// TIA Portal project "激光打标_V15.1" (V15.1)

(* hardware
DEVICE "S7-1200 station_1"  S7-1200 Station
   slot 0: "Rack_0"  S7-1200 Rack  Rack  V1.0
   slot 1: "A170648_14 CPU  1214C"  CPU 1214C DC/DC/DC  6ES7 214-1AG40-0XB0  V4.2
   slot 2: "DI 16x24VDC/DQ 16xRelay_1"  SM 1223 DI16/DQ16 x relay  6ES7 223-1PL32-0XB0  V2.0
   slot 3: "DI 16x24VDC/DQ 16xRelay_2"  SM 1223 DI16/DQ16 x relay  6ES7 223-1PL32-0XB0  V2.0
*)

// ===== PLC "A170648_14 CPU  1214C"  CPU 1214C DC/DC/DC =====

VAR_GLOBAL   // PLC tag table "默认变量表"
   "启动" AT %I0.0 : Bool;
   "复位" AT %I0.1 : Bool;
   "安全门" AT %I0.2 : Bool;
   "急停" AT %I0.3 : Bool;
   "气源检测" AT %I0.4 : Bool;
   "手自动" AT %I0.5 : Bool;
   "激光打码完成" AT %I0.6 : Bool;
   "激光打码报警" AT %I0.7 : Bool;
   "1#升降按钮" AT %I1.0 : Bool;
   "1#气爪松紧按钮" AT %I1.1 : Bool;
   "1#固定按钮" AT %I1.2 : Bool;
   "2#升降按钮" AT %I1.3 : Bool;
   "2#气爪松紧按钮" AT %I1.4 : Bool;
   "2#固定按钮" AT %I1.5 : Bool;
   "工件在位" AT %I2.0 : Bool;
   "防护门上限位" AT %I2.1 : Bool;
   "防护门下限位" AT %I2.2 : Bool;
   "工装移栽进到位" AT %I2.3 : Bool;
   "工装移栽退到位" AT %I2.4 : Bool;
   "备用(2)" AT %I2.5 : Bool;
   "备用(4)" AT %I2.6 : Bool;
   "备用(3)" AT %I2.7 : Bool;
   "1#固定进到位" AT %I3.0 : Bool;
   "1#固定退到位" AT %I3.1 : Bool;
   "备用" AT %I3.2 : Bool;
   "1#左气爪松开到位" AT %I3.3 : Bool;
   "备用(1)" AT %I3.4 : Bool;
   "1#右气爪松开到位" AT %I3.5 : Bool;
   "1#机械手升到位" AT %I3.6 : Bool;
   "1#机械手降到位" AT %I3.7 : Bool;
   "2#机械手升到位" AT %I4.0 : Bool;
   "2#机械手降到位" AT %I4.1 : Bool;
   "备用(31)" AT %I4.2 : Bool;
   "2#左气爪松开到位" AT %I4.3 : Bool;
   "备用(32)" AT %I4.4 : Bool;
   "2#右气爪松开到位" AT %I4.5 : Bool;
   "2#固定进到位" AT %I4.6 : Bool;
   "2#固定退到位" AT %I4.7 : Bool;
   "备用(5)" AT %I5.0 : Bool;
   "备用(6)" AT %I5.1 : Bool;
   "备用(7)" AT %I5.2 : Bool;
   "备用(8)" AT %I5.3 : Bool;
   "备用(9)" AT %I5.4 : Bool;
   "备用(10)" AT %I5.5 : Bool;
   "备用(11)" AT %I5.6 : Bool;
   "备用(12)" AT %I5.7 : Bool;
   "启动打标" AT %Q0.0 : Bool;
   "备用(13)" AT %Q0.1 : Bool;
   "三色灯——红" AT %Q0.2 : Bool;
   "三色灯——黄" AT %Q0.3 : Bool;
   "三色灯——绿" AT %Q0.4 : Bool;
   "三色灯——蜂鸣器" AT %Q0.5 : Bool;
   "气源开关" AT %Q0.6 : Bool;
   "备用(14)" AT %Q0.7 : Bool;
   "合格指示灯" AT %Q1.0 : Bool;
   "不合格指示灯" AT %Q1.1 : Bool;
   "防护门上升" AT %Q2.0 : Bool;
   "防护门下降" AT %Q2.1 : Bool;
   "工装移载前进" AT %Q2.2 : Bool;
   "工装移载后退" AT %Q2.3 : Bool;
   "备用(15)" AT %Q2.4 : Bool;
   "备用(16)" AT %Q2.5 : Bool;
   "备用(17)" AT %Q2.6 : Bool;
   "备用(18)" AT %Q2.7 : Bool;
   "1#机械手上升" AT %Q3.0 : Bool;
   "1#机械手下降" AT %Q3.1 : Bool;
   "1#机械手气爪夹紧" AT %Q3.2 : Bool;
   "1#机械手气爪松开" AT %Q3.3 : Bool;
   "备用(19)" AT %Q3.4 : Bool;
   "备用(20)" AT %Q3.5 : Bool;
   "1#固定气缸进" AT %Q3.6 : Bool;
   "1#固定气缸退" AT %Q3.7 : Bool;
   "2#机械手上升" AT %Q4.0 : Bool;
   "2#机械手下降" AT %Q4.1 : Bool;
   "2#机械手气爪夹紧" AT %Q4.2 : Bool;
   "2#机械手气爪松开" AT %Q4.3 : Bool;
   "备用(21)" AT %Q4.4 : Bool;
   "备用(22)" AT %Q4.5 : Bool;
   "2#固定气缸进" AT %Q4.6 : Bool;
   "2#固定气缸退" AT %Q4.7 : Bool;
   "备用(23)" AT %Q5.0 : Bool;
   "备用(24)" AT %Q5.1 : Bool;
   "备用(25)" AT %Q5.2 : Bool;
   "备用(26)" AT %Q5.3 : Bool;
   "备用(27)" AT %Q5.4 : Bool;
   "备用(28)" AT %Q5.5 : Bool;
   "备用(29)" AT %Q5.6 : Bool;
   "备用(30)" AT %Q5.7 : Bool;
   "程序停止" AT %M100.0 : Bool;
   "复位完成" AT %M100.1 : Bool;
   "Clock_1Hz" AT %M0.5 : Bool;
   "Tag_1" AT %M100.3 : Bool;
   "AlwaysFALSE" AT %M1.3 : Bool;
   "Tag_2" AT %M30.0 : Bool;
   "Clock_Byte" AT %MB0 : Byte;
   "Clock_10Hz" AT %M0.0 : Bool;
   "Clock_5Hz" AT %M0.1 : Bool;
   "Clock_2.5Hz" AT %M0.2 : Bool;
   "Clock_2Hz" AT %M0.3 : Bool;
   "Clock_1.25Hz" AT %M0.4 : Bool;
   "Clock_0.625Hz" AT %M0.6 : Bool;
   "Clock_0.5Hz" AT %M0.7 : Bool;
   "System_Byte" AT %MB1 : Byte;
   "FirstScan" AT %M1.0 : Bool;
   "DiagStatusUpdate" AT %M1.1 : Bool;
   "AlwaysTRUE" AT %M1.2 : Bool;
   "Tag_3" AT %M300.0 : Bool;
   "Tag_4" AT %M300.4 : Bool;
   "Tag_5" AT %M300.1 : Bool;
   "Tag_6" AT %M300.5 : Bool;
   "Tag_7" AT %M300.3 : Bool;
   "Tag_8" AT %M300.7 : Bool;
   "Tag_9" AT %M312.0 : Bool;
   "Tag_10" AT %M3000.0 : Bool;
   "Tag_11" AT %M3000.1 : Bool;
   "Tag_12" AT %MD3004 : DWord;
   "Tag_13" AT %M3000.2 : Bool;
   "Tag_14" AT %M3000.3 : Bool;
   "Tag_15" AT %MW3004 : Word;
   "Tag_16" AT %M312.1 : Bool;
   "Tag_17" AT %M200.0 : Bool;
   "Tag_18" AT %M200.6 : Bool;
   "Tag_19" AT %M200.7 : Bool;
   "吸尘器" AT %MB10 : SInt;
END_VAR

DATA_BLOCK "SERVER"   // DB1
{ S7_Optimized_Access := 'FALSE' }
VERSION : 0.1
   VAR
      设备状态 : Int := 0;
      产品型号 : Int := 0;
      错误代码 : Int := 0;
      生产结果 : Int := 0;
      设备编号 : Int := 0;
      吸尘器 : Int;
   END_VAR
BEGIN
END_DATA_BLOCK

DATA_BLOCK "MB_TCON"   // DB2
{ S7_Optimized_Access := 'FALSE' }
VERSION : 0.1
   VAR
      MB_TCON : TCON_IP_v4;
   END_VAR
BEGIN
   MB_TCON.InterfaceId := 64;
   MB_TCON.ID := 1;
   MB_TCON.LocalPort := 502;
   MB_TCON.RemoteAddress.ADDR[1] := 0;
   MB_TCON.RemoteAddress.ADDR[2] := 0;
   MB_TCON.RemoteAddress.ADDR[3] := 0;
   MB_TCON.RemoteAddress.ADDR[4] := 0;
END_DATA_BLOCK

DATA_BLOCK "RESET_DB"   // DB3
{ S7_Optimized_Access := 'TRUE' }
VERSION : 0.1
// stored: InstanceOfName RESET
"RESET"
BEGIN
END_DATA_BLOCK

DATA_BLOCK "ALARM_DB"   // DB4
{ S7_Optimized_Access := 'TRUE' }
VERSION : 0.1
// stored: InstanceOfName ALARM
"ALARM"
BEGIN
END_DATA_BLOCK

DATA_BLOCK "1# jixieshou_DB"   // DB8
{ S7_Optimized_Access := 'TRUE' }
VERSION : 0.1
// stored: InstanceOfName 1# jixieshou
"1# jixieshou"
BEGIN
END_DATA_BLOCK

DATA_BLOCK "2#jixieshou_DB"   // DB9
{ S7_Optimized_Access := 'TRUE' }
VERSION : 0.1
// stored: InstanceOfName 2#jixieshou
"2#jixieshou"
BEGIN
END_DATA_BLOCK

DATA_BLOCK "AUTO_DB"   // DB10
{ S7_Optimized_Access := 'TRUE' }
VERSION : 0.1
// stored: InstanceOfName AUTO
"AUTO"
BEGIN
END_DATA_BLOCK

// folder: System blocks/Program resources

DATA_BLOCK "IEC_Timer_0_DB"   // DB5
{ S7_Optimized_Access := 'TRUE' }
AUTHOR : Simatic
FAMILY : IEC
NAME : IEC_TMR
VERSION : 1.0
// stored: InstanceOfName IEC_TIMER
"IEC_TIMER"
BEGIN
END_DATA_BLOCK

DATA_BLOCK "IEC_Timer_0_DB_1"   // DB6
{ S7_Optimized_Access := 'TRUE' }
AUTHOR : Simatic
FAMILY : IEC
NAME : IEC_TMR
VERSION : 1.0
// stored: InstanceOfName IEC_TIMER
"IEC_TIMER"
BEGIN
END_DATA_BLOCK

DATA_BLOCK "IEC_Timer_0_DB_3"   // DB12
{ S7_Optimized_Access := 'TRUE' }
AUTHOR : Simatic
FAMILY : IEC
NAME : IEC_TMR
VERSION : 1.0
// stored: InstanceOfName IEC_TIMER
"IEC_TIMER"
BEGIN
END_DATA_BLOCK

// folder: (top level)

FUNCTION_BLOCK "ALARM"   // FB1, LAD
{ S7_Optimized_Access := 'TRUE' }
VERSION : 0.1
   VAR
      "Error-ID" : Word;
      TEmp : Array[0..3] of Bool;
      IEC_Timer_0_Instance : TON_TIME;
      IEC_Timer_0_Instance_1 : TON_TIME;
      IEC_Timer_0_Instance_2 : TON_TIME;
      IEC_Timer_0_Instance_3 : TON_TIME;
      IEC_Timer_0_Instance_4 : TON_TIME;
      IEC_Timer_0_Instance_5 : TON_TIME;
      IEC_Timer_0_Instance_6 : TON_TIME;
      IEC_Timer_0_Instance_7 : TON_TIME;
      IEC_Timer_0_Instance_8 : TON_TIME;
      IEC_Timer_0_Instance_9 : TON_TIME;
      IEC_Timer_0_Instance_10 : TON_TIME;
      IEC_Timer_0_Instance_11 : TON_TIME;
      IEC_Timer_0_Instance_12 : TON_TIME;
      IEC_Timer_0_Instance_13 : TON_TIME;
      IEC_Timer_0_Instance_14 : TON_TIME;
      "STEP" : Int;
      IEC_Timer_0_Instance_15 : TON_TIME;
      IEC_Timer_0_Instance_16 : TON_TIME;
   END_VAR
   VAR_TEMP   // added for the SCL form of the ladder/FBD networks
      _w1 : Bool;
   END_VAR
BEGIN

REGION Network 1
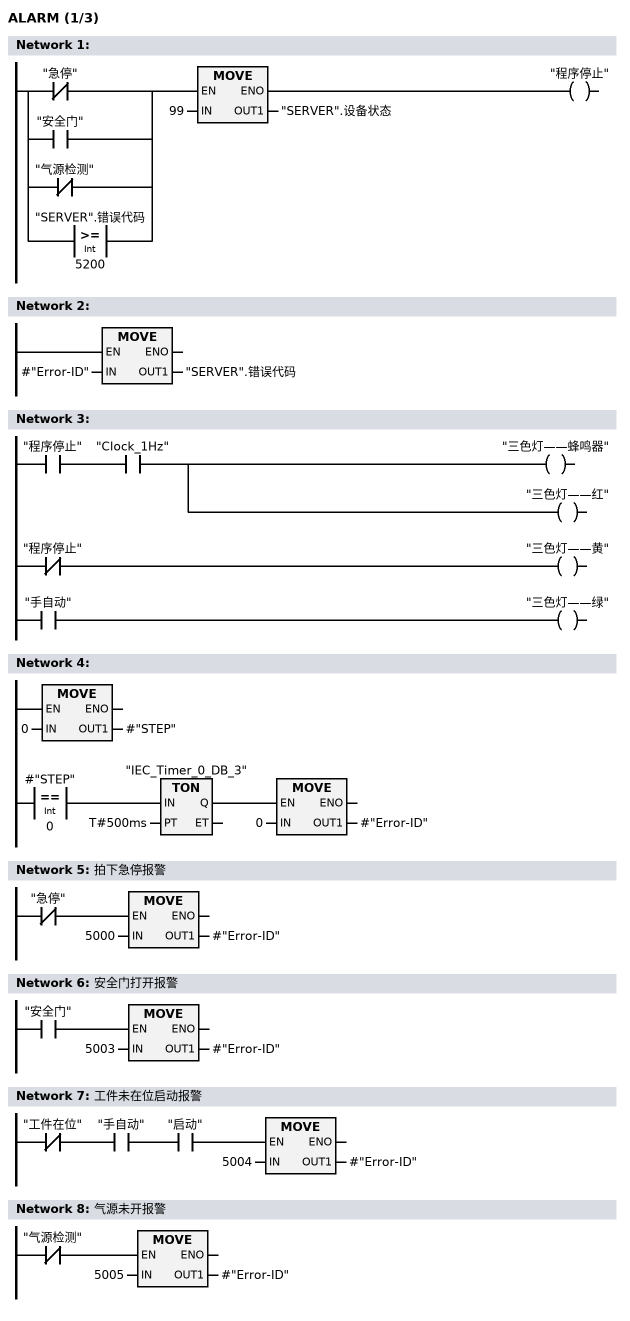
   RUNG wire#powerrail
      I_Contact( "急停" )
      wire#w1
      Move(in := 99, out1 => "SERVER".设备状态)
      Coil( "程序停止" )
   END_RUNG
   RUNG wire#powerrail
      Contact( "安全门" )
   END_RUNG wire#w1
   RUNG wire#powerrail
      I_Contact( "气源检测" )
   END_RUNG wire#w1
   RUNG wire#powerrail
      { S7_Templates := "SrcType := Int" } GE_Contact(in1 := "SERVER".错误代码, in2 := 5200)
   END_RUNG wire#w1
   // the same network as SCL:
   #_w1 := NOT "急停" OR "安全门" OR NOT "气源检测" OR ("SERVER".错误代码 >= 5200);
   IF #_w1 THEN "SERVER".设备状态 := 99; END_IF;
   "程序停止" := #_w1;
END_REGION

REGION Network 2
   RUNG wire#powerrail
      Move(in := #"Error-ID", out1 => "SERVER".错误代码)
   END_RUNG
   // the same network as SCL:
   "SERVER".错误代码 := #"Error-ID";
END_REGION

REGION Network 3
   RUNG wire#powerrail
      Contact( "程序停止" )
      Contact( "Clock_1Hz" )
      wire#w1
      Coil( "三色灯——蜂鸣器" )
   END_RUNG
   RUNG wire#w1
      Coil( "三色灯——红" )
   END_RUNG
   RUNG wire#powerrail
      I_Contact( "程序停止" )
      Coil( "三色灯——黄" )
   END_RUNG
   RUNG wire#powerrail
      Contact( "手自动" )
      Coil( "三色灯——绿" )
   END_RUNG
   // the same network as SCL:
   "三色灯——蜂鸣器" := "程序停止" AND "Clock_1Hz";
   "三色灯——红" := "三色灯——蜂鸣器";
   "三色灯——黄" := NOT "程序停止";
   "三色灯——绿" := "手自动";
END_REGION

REGION Network 4
   #"STEP" := 0;
   "IEC_Timer_0_DB_3".TON(IN := #"STEP" = 0, PT := T#500ms);
   IF "IEC_Timer_0_DB_3".Q THEN #"Error-ID" := 0; END_IF;
END_REGION

REGION Network 5: 拍下急停报警
   RUNG wire#powerrail
      I_Contact( "急停" )
      Move(in := 5000, out1 => #"Error-ID")
   END_RUNG
   // the same network as SCL:
   IF NOT "急停" THEN #"Error-ID" := 5000; END_IF;
END_REGION

REGION Network 6: 安全门打开报警
   RUNG wire#powerrail
      Contact( "安全门" )
      Move(in := 5003, out1 => #"Error-ID")
   END_RUNG
   // the same network as SCL:
   IF "安全门" THEN #"Error-ID" := 5003; END_IF;
END_REGION

REGION Network 7: 工件未在位启动报警
   RUNG wire#powerrail
      I_Contact( "工件在位" )
      Contact( "手自动" )
      Contact( "启动" )
      Move(in := 5004, out1 => #"Error-ID")
   END_RUNG
   // the same network as SCL:
   IF NOT "工件在位" AND "手自动" AND "启动" THEN #"Error-ID" := 5004; END_IF;
END_REGION

REGION Network 8: 气源未开报警
   RUNG wire#powerrail
      I_Contact( "气源检测" )
      Move(in := 5005, out1 => #"Error-ID")
   END_RUNG
   // the same network as SCL:
   IF NOT "气源检测" THEN #"Error-ID" := 5005; END_IF;
END_REGION

REGION Network 9: 工装移栽前进未到位报警
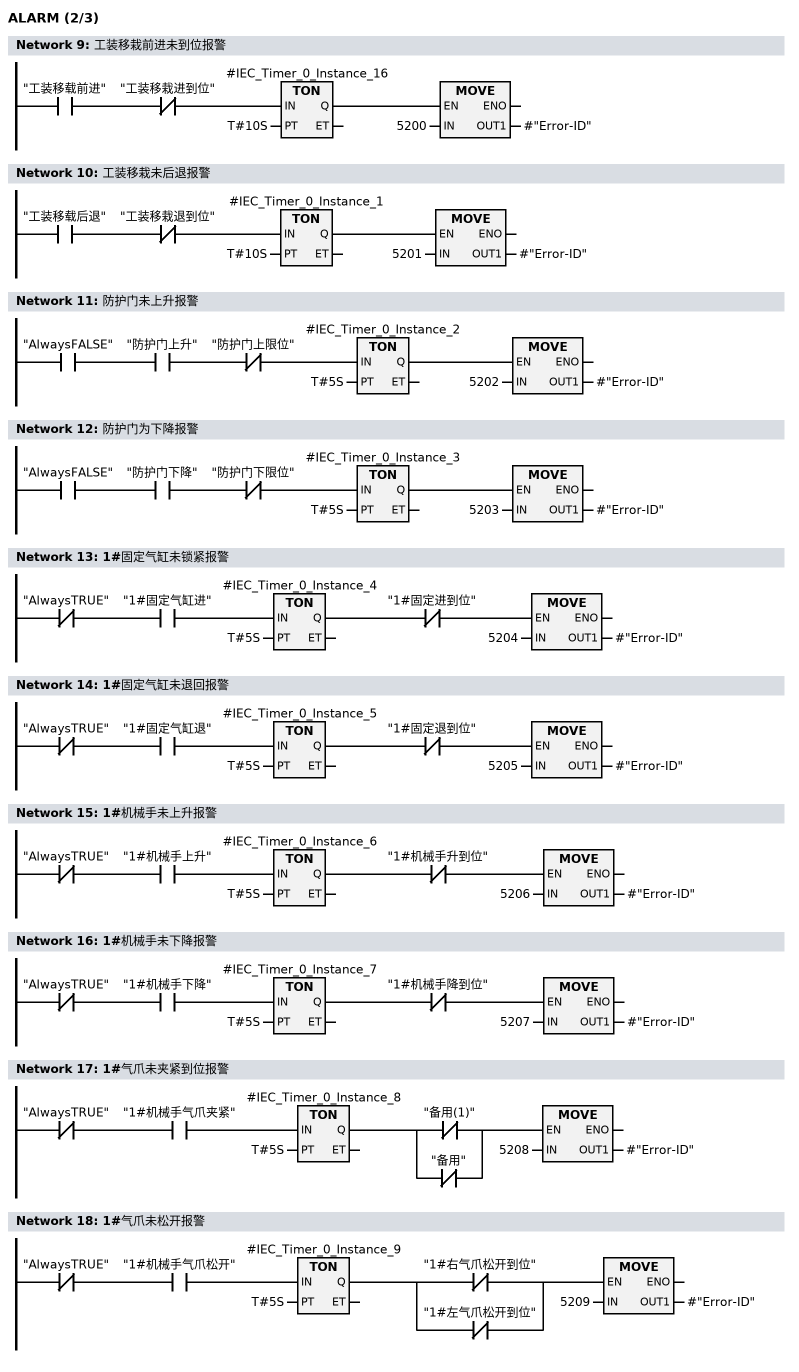
   #IEC_Timer_0_Instance_16(IN := "工装移载前进" AND NOT "工装移栽进到位", PT := T#10S);   // TON
   IF #IEC_Timer_0_Instance_16.Q THEN #"Error-ID" := 5200; END_IF;
END_REGION

REGION Network 10: 工装移栽未后退报警
   #IEC_Timer_0_Instance_1(IN := "工装移载后退" AND NOT "工装移栽退到位", PT := T#10S);   // TON
   IF #IEC_Timer_0_Instance_1.Q THEN #"Error-ID" := 5201; END_IF;
END_REGION

REGION Network 11: 防护门未上升报警
   #IEC_Timer_0_Instance_2(IN := "AlwaysFALSE" AND "防护门上升" AND NOT "防护门上限位", PT := T#5S);   // TON
   IF #IEC_Timer_0_Instance_2.Q THEN #"Error-ID" := 5202; END_IF;
END_REGION

REGION Network 12: 防护门为下降报警
   #IEC_Timer_0_Instance_3(IN := "AlwaysFALSE" AND "防护门下降" AND NOT "防护门下限位", PT := T#5S);   // TON
   IF #IEC_Timer_0_Instance_3.Q THEN #"Error-ID" := 5203; END_IF;
END_REGION

REGION Network 13: 1#固定气缸未锁紧报警
   #IEC_Timer_0_Instance_4(IN := NOT "AlwaysTRUE" AND "1#固定气缸进", PT := T#5S);   // TON
   IF #IEC_Timer_0_Instance_4.Q AND NOT "1#固定进到位" THEN #"Error-ID" := 5204; END_IF;
END_REGION

REGION Network 14: 1#固定气缸未退回报警
   #IEC_Timer_0_Instance_5(IN := NOT "AlwaysTRUE" AND "1#固定气缸退", PT := T#5S);   // TON
   IF #IEC_Timer_0_Instance_5.Q AND NOT "1#固定退到位" THEN #"Error-ID" := 5205; END_IF;
END_REGION

REGION Network 15: 1#机械手未上升报警
   #IEC_Timer_0_Instance_6(IN := NOT "AlwaysTRUE" AND "1#机械手上升", PT := T#5S);   // TON
   IF #IEC_Timer_0_Instance_6.Q AND NOT "1#机械手升到位" THEN #"Error-ID" := 5206; END_IF;
END_REGION

REGION Network 16: 1#机械手未下降报警
   #IEC_Timer_0_Instance_7(IN := NOT "AlwaysTRUE" AND "1#机械手下降", PT := T#5S);   // TON
   IF #IEC_Timer_0_Instance_7.Q AND NOT "1#机械手降到位" THEN #"Error-ID" := 5207; END_IF;
END_REGION

REGION Network 17: 1#气爪未夹紧到位报警
   #IEC_Timer_0_Instance_8(IN := NOT "AlwaysTRUE" AND "1#机械手气爪夹紧", PT := T#5S);   // TON
   IF #IEC_Timer_0_Instance_8.Q AND (NOT "备用(1)" OR NOT "备用") THEN #"Error-ID" := 5208; END_IF;
END_REGION

REGION Network 18: 1#气爪未松开报警
   #IEC_Timer_0_Instance_9(IN := NOT "AlwaysTRUE" AND "1#机械手气爪松开", PT := T#5S);   // TON
   IF #IEC_Timer_0_Instance_9.Q AND (NOT "1#右气爪松开到位" OR NOT "1#左气爪松开到位") THEN #"Error-ID" := 5209; END_IF;
END_REGION

REGION Network 19: 2#机械手未固定锁紧报警
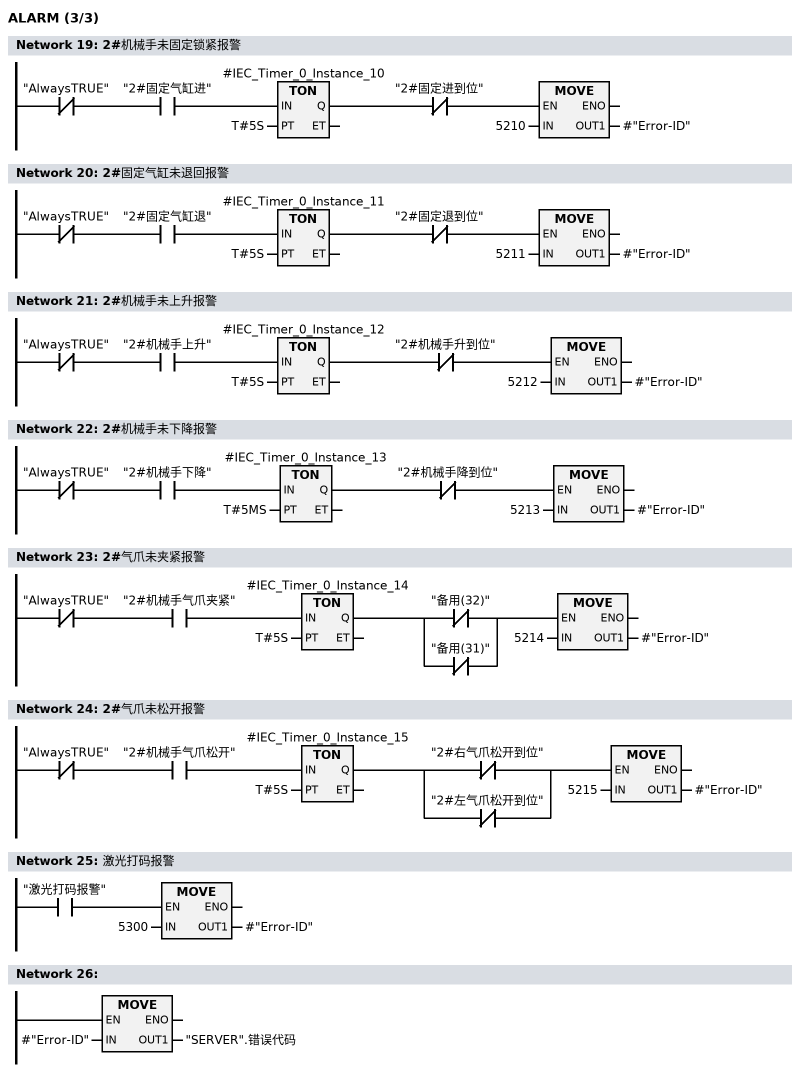
   #IEC_Timer_0_Instance_10(IN := NOT "AlwaysTRUE" AND "2#固定气缸进", PT := T#5S);   // TON
   IF #IEC_Timer_0_Instance_10.Q AND NOT "2#固定进到位" THEN #"Error-ID" := 5210; END_IF;
END_REGION

REGION Network 20: 2#固定气缸未退回报警
   #IEC_Timer_0_Instance_11(IN := NOT "AlwaysTRUE" AND "2#固定气缸退", PT := T#5S);   // TON
   IF #IEC_Timer_0_Instance_11.Q AND NOT "2#固定退到位" THEN #"Error-ID" := 5211; END_IF;
END_REGION

REGION Network 21: 2#机械手未上升报警
   #IEC_Timer_0_Instance_12(IN := NOT "AlwaysTRUE" AND "2#机械手上升", PT := T#5S);   // TON
   IF #IEC_Timer_0_Instance_12.Q AND NOT "2#机械手升到位" THEN #"Error-ID" := 5212; END_IF;
END_REGION

REGION Network 22: 2#机械手未下降报警
   #IEC_Timer_0_Instance_13(IN := NOT "AlwaysTRUE" AND "2#机械手下降", PT := T#5MS);   // TON
   IF #IEC_Timer_0_Instance_13.Q AND NOT "2#机械手降到位" THEN #"Error-ID" := 5213; END_IF;
END_REGION

REGION Network 23: 2#气爪未夹紧报警
   #IEC_Timer_0_Instance_14(IN := NOT "AlwaysTRUE" AND "2#机械手气爪夹紧", PT := T#5S);   // TON
   IF #IEC_Timer_0_Instance_14.Q AND (NOT "备用(32)" OR NOT "备用(31)") THEN #"Error-ID" := 5214; END_IF;
END_REGION

REGION Network 24: 2#气爪未松开报警
   #IEC_Timer_0_Instance_15(IN := NOT "AlwaysTRUE" AND "2#机械手气爪松开", PT := T#5S);   // TON
   IF #IEC_Timer_0_Instance_15.Q AND (NOT "2#右气爪松开到位" OR NOT "2#左气爪松开到位") THEN #"Error-ID" := 5215; END_IF;
END_REGION

REGION Network 25: 激光打码报警
   RUNG wire#powerrail
      Contact( "激光打码报警" )
      Move(in := 5300, out1 => #"Error-ID")
   END_RUNG
   // the same network as SCL:
   IF "激光打码报警" THEN #"Error-ID" := 5300; END_IF;
END_REGION

REGION Network 26
   RUNG wire#powerrail
      Move(in := #"Error-ID", out1 => "SERVER".错误代码)
   END_RUNG
   // the same network as SCL:
   "SERVER".错误代码 := #"Error-ID";
END_REGION
END_FUNCTION_BLOCK

FUNCTION_BLOCK "RESET"   // FB2, LAD
{ S7_Optimized_Access := 'TRUE' }
VERSION : 0.1
   VAR_INPUT
      Stop : Bool;
      Start : Bool;
   END_VAR
   VAR_OUTPUT
      Down : Bool;
   END_VAR
   VAR
      "Step" : Int;
   END_VAR
   VAR_TEMP   // added for the SCL form of the ladder/FBD networks
      _w1 : Bool;
   END_VAR
BEGIN

REGION Network 1
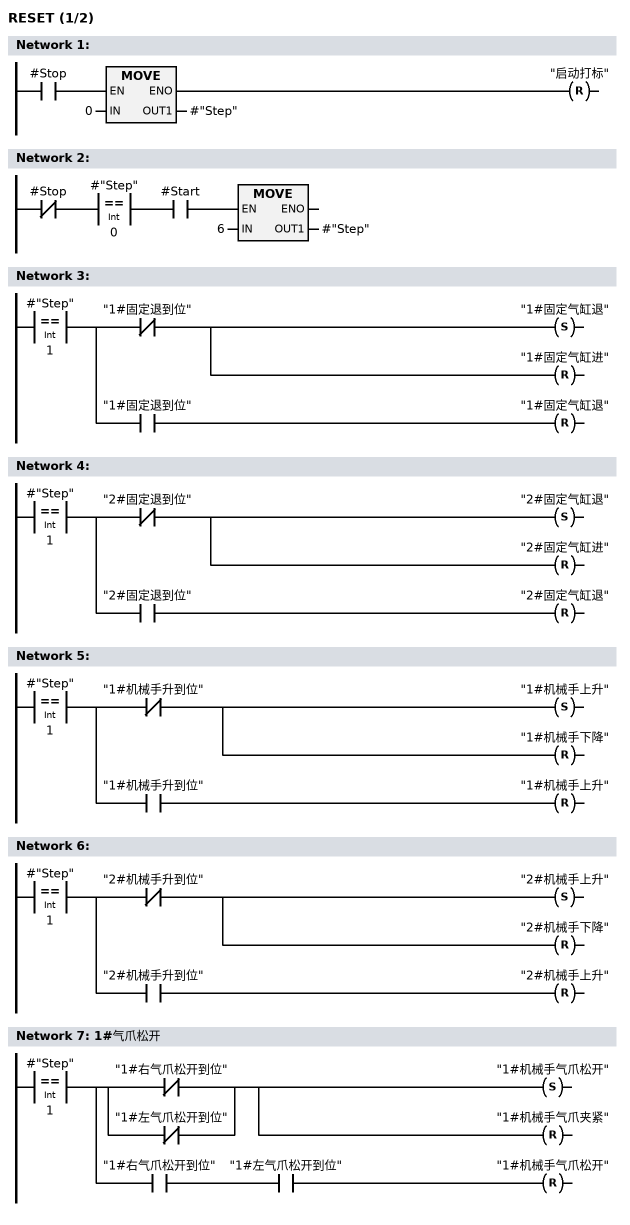
   RUNG wire#powerrail
      Contact( #Stop )
      Move(in := 0, out1 => #"Step")
      R_Coil( "启动打标" )
   END_RUNG
   // the same network as SCL:
   IF #Stop THEN
       #"Step" := 0;
       "启动打标" := FALSE;
   END_IF;
END_REGION

REGION Network 2
   RUNG wire#powerrail
      I_Contact( #Stop )
      { S7_Templates := "SrcType := Int" } EQ_Contact(in1 := #"Step", in2 := 0)
      Contact( #Start )
      Move(in := 6, out1 => #"Step")
   END_RUNG
   // the same network as SCL:
   IF NOT #Stop AND (#"Step" = 0) AND #Start THEN #"Step" := 6; END_IF;
END_REGION

REGION Network 3
   RUNG wire#powerrail
      { S7_Templates := "SrcType := Int" } EQ_Contact(in1 := #"Step", in2 := 1)
      wire#w1
      I_Contact( "1#固定退到位" )
      wire#w2
      S_Coil( "1#固定气缸退" )
   END_RUNG
   RUNG wire#w2
      R_Coil( "1#固定气缸进" )
   END_RUNG
   RUNG wire#w1
      Contact( "1#固定退到位" )
      R_Coil( "1#固定气缸退" )
   END_RUNG
   // the same network as SCL:
   #_w1 := #"Step" = 1;
   IF #_w1 AND NOT "1#固定退到位" THEN
       "1#固定气缸退" := TRUE;
       "1#固定气缸进" := FALSE;
   END_IF;
   IF #_w1 AND "1#固定退到位" THEN "1#固定气缸退" := FALSE; END_IF;
END_REGION

REGION Network 4
   RUNG wire#powerrail
      { S7_Templates := "SrcType := Int" } EQ_Contact(in1 := #"Step", in2 := 1)
      wire#w1
      I_Contact( "2#固定退到位" )
      wire#w2
      S_Coil( "2#固定气缸退" )
   END_RUNG
   RUNG wire#w2
      R_Coil( "2#固定气缸进" )
   END_RUNG
   RUNG wire#w1
      Contact( "2#固定退到位" )
      R_Coil( "2#固定气缸退" )
   END_RUNG
   // the same network as SCL:
   #_w1 := #"Step" = 1;
   IF #_w1 AND NOT "2#固定退到位" THEN
       "2#固定气缸退" := TRUE;
       "2#固定气缸进" := FALSE;
   END_IF;
   IF #_w1 AND "2#固定退到位" THEN "2#固定气缸退" := FALSE; END_IF;
END_REGION

REGION Network 5
   RUNG wire#powerrail
      { S7_Templates := "SrcType := Int" } EQ_Contact(in1 := #"Step", in2 := 1)
      wire#w1
      I_Contact( "1#机械手升到位" )
      wire#w2
      S_Coil( "1#机械手上升" )
   END_RUNG
   RUNG wire#w2
      R_Coil( "1#机械手下降" )
   END_RUNG
   RUNG wire#w1
      Contact( "1#机械手升到位" )
      R_Coil( "1#机械手上升" )
   END_RUNG
   // the same network as SCL:
   #_w1 := #"Step" = 1;
   IF #_w1 AND NOT "1#机械手升到位" THEN
       "1#机械手上升" := TRUE;
       "1#机械手下降" := FALSE;
   END_IF;
   IF #_w1 AND "1#机械手升到位" THEN "1#机械手上升" := FALSE; END_IF;
END_REGION

REGION Network 6
   RUNG wire#powerrail
      { S7_Templates := "SrcType := Int" } EQ_Contact(in1 := #"Step", in2 := 1)
      wire#w1
      I_Contact( "2#机械手升到位" )
      wire#w2
      S_Coil( "2#机械手上升" )
   END_RUNG
   RUNG wire#w2
      R_Coil( "2#机械手下降" )
   END_RUNG
   RUNG wire#w1
      Contact( "2#机械手升到位" )
      R_Coil( "2#机械手上升" )
   END_RUNG
   // the same network as SCL:
   #_w1 := #"Step" = 1;
   IF #_w1 AND NOT "2#机械手升到位" THEN
       "2#机械手上升" := TRUE;
       "2#机械手下降" := FALSE;
   END_IF;
   IF #_w1 AND "2#机械手升到位" THEN "2#机械手上升" := FALSE; END_IF;
END_REGION

REGION Network 7: 1#气爪松开
   RUNG wire#powerrail
      { S7_Templates := "SrcType := Int" } EQ_Contact(in1 := #"Step", in2 := 1)
      wire#w1
      I_Contact( "1#右气爪松开到位" )
      wire#w2
      S_Coil( "1#机械手气爪松开" )
   END_RUNG
   RUNG wire#w1
      I_Contact( "1#左气爪松开到位" )
   END_RUNG wire#w2
   RUNG wire#w2
      R_Coil( "1#机械手气爪夹紧" )
   END_RUNG
   RUNG wire#w1
      Contact( "1#右气爪松开到位" )
      Contact( "1#左气爪松开到位" )
      R_Coil( "1#机械手气爪松开" )
   END_RUNG
   // the same network as SCL:
   #_w1 := #"Step" = 1;
   IF #_w1 AND (NOT "1#右气爪松开到位" OR NOT "1#左气爪松开到位") THEN
       "1#机械手气爪松开" := TRUE;
       "1#机械手气爪夹紧" := FALSE;
   END_IF;
   IF #_w1 AND "1#右气爪松开到位" AND "1#左气爪松开到位" THEN "1#机械手气爪松开" := FALSE; END_IF;
END_REGION

REGION Network 8: 2#气爪松开
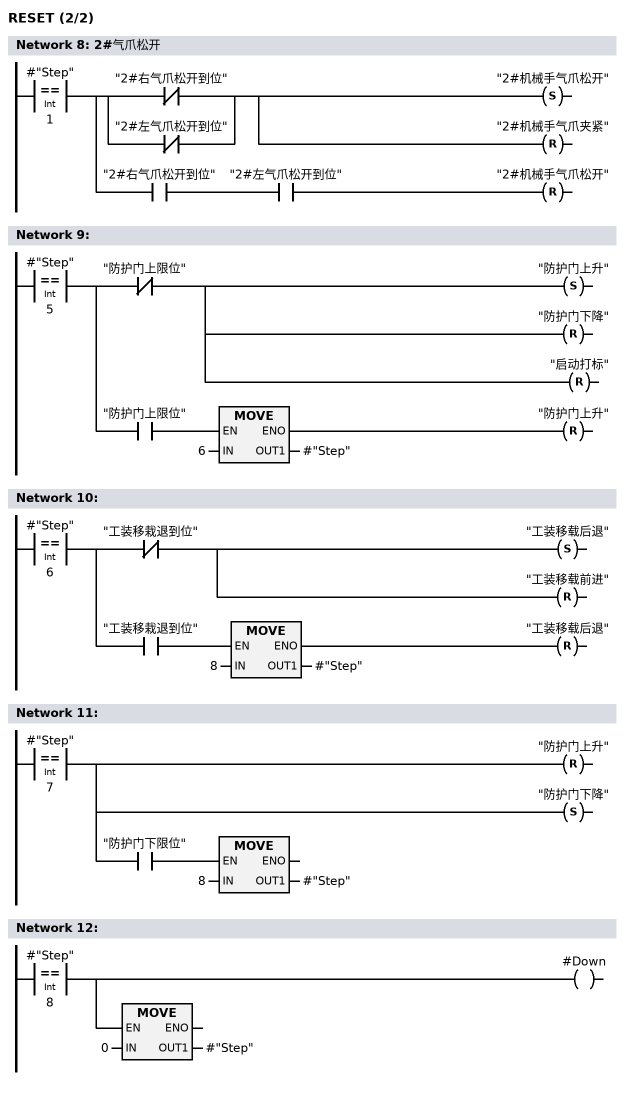
   RUNG wire#powerrail
      { S7_Templates := "SrcType := Int" } EQ_Contact(in1 := #"Step", in2 := 1)
      wire#w1
      I_Contact( "2#右气爪松开到位" )
      wire#w2
      S_Coil( "2#机械手气爪松开" )
   END_RUNG
   RUNG wire#w1
      I_Contact( "2#左气爪松开到位" )
   END_RUNG wire#w2
   RUNG wire#w2
      R_Coil( "2#机械手气爪夹紧" )
   END_RUNG
   RUNG wire#w1
      Contact( "2#右气爪松开到位" )
      Contact( "2#左气爪松开到位" )
      R_Coil( "2#机械手气爪松开" )
   END_RUNG
   // the same network as SCL:
   #_w1 := #"Step" = 1;
   IF #_w1 AND (NOT "2#右气爪松开到位" OR NOT "2#左气爪松开到位") THEN
       "2#机械手气爪松开" := TRUE;
       "2#机械手气爪夹紧" := FALSE;
   END_IF;
   IF #_w1 AND "2#右气爪松开到位" AND "2#左气爪松开到位" THEN "2#机械手气爪松开" := FALSE; END_IF;
END_REGION

REGION Network 9
   RUNG wire#powerrail
      { S7_Templates := "SrcType := Int" } EQ_Contact(in1 := #"Step", in2 := 5)
      wire#w1
      I_Contact( "防护门上限位" )
      wire#w2
      S_Coil( "防护门上升" )
   END_RUNG
   RUNG wire#w2
      R_Coil( "防护门下降" )
   END_RUNG
   RUNG wire#w2
      R_Coil( "启动打标" )
   END_RUNG
   RUNG wire#w1
      Contact( "防护门上限位" )
      Move(in := 6, out1 => #"Step")
      R_Coil( "防护门上升" )
   END_RUNG
   // the same network as SCL:
   #_w1 := #"Step" = 5;
   IF #_w1 AND NOT "防护门上限位" THEN
       "防护门上升" := TRUE;
       "防护门下降" := FALSE;
       "启动打标" := FALSE;
   END_IF;
   IF #_w1 AND "防护门上限位" THEN
       #"Step" := 6;
       "防护门上升" := FALSE;
   END_IF;
END_REGION

REGION Network 10
   RUNG wire#powerrail
      { S7_Templates := "SrcType := Int" } EQ_Contact(in1 := #"Step", in2 := 6)
      wire#w1
      I_Contact( "工装移栽退到位" )
      wire#w2
      S_Coil( "工装移载后退" )
   END_RUNG
   RUNG wire#w2
      R_Coil( "工装移载前进" )
   END_RUNG
   RUNG wire#w1
      Contact( "工装移栽退到位" )
      Move(in := 8, out1 => #"Step")
      R_Coil( "工装移载后退" )
   END_RUNG
   // the same network as SCL:
   #_w1 := #"Step" = 6;
   IF #_w1 AND NOT "工装移栽退到位" THEN
       "工装移载后退" := TRUE;
       "工装移载前进" := FALSE;
   END_IF;
   IF #_w1 AND "工装移栽退到位" THEN
       #"Step" := 8;
       "工装移载后退" := FALSE;
   END_IF;
END_REGION

REGION Network 11
   RUNG wire#powerrail
      { S7_Templates := "SrcType := Int" } EQ_Contact(in1 := #"Step", in2 := 7)
      wire#w1
      R_Coil( "防护门上升" )
   END_RUNG
   RUNG wire#w1
      S_Coil( "防护门下降" )
   END_RUNG
   RUNG wire#w1
      Contact( "防护门下限位" )
      Move(in := 8, out1 => #"Step")
   END_RUNG
   // the same network as SCL:
   #_w1 := #"Step" = 7;
   IF #_w1 THEN
       "防护门上升" := FALSE;
       "防护门下降" := TRUE;
   END_IF;
   IF #_w1 AND "防护门下限位" THEN #"Step" := 8; END_IF;
END_REGION

REGION Network 12
   RUNG wire#powerrail
      { S7_Templates := "SrcType := Int" } EQ_Contact(in1 := #"Step", in2 := 8)
      wire#w1
      Coil( #Down )
   END_RUNG
   RUNG wire#w1
      Move(in := 0, out1 => #"Step")
   END_RUNG
   // the same network as SCL:
   #Down := #"Step" = 8;
   IF #Down THEN #"Step" := 0; END_IF;
END_REGION
END_FUNCTION_BLOCK

FUNCTION_BLOCK "AUTO"   // FB3, LAD
{ S7_Optimized_Access := 'TRUE' }
VERSION : 0.1
   VAR
      IEC_Timer_0_Instance : TON_TIME;
      IEC_Timer_0_Instance_1 : TON_TIME;
      IEC_Timer_0_Instance_2 : TON_TIME;
   END_VAR
   VAR_TEMP   // added for the SCL form of the ladder/FBD networks
      _w1 : Bool;
      _w2 : Bool;
   END_VAR
BEGIN

REGION Network 1
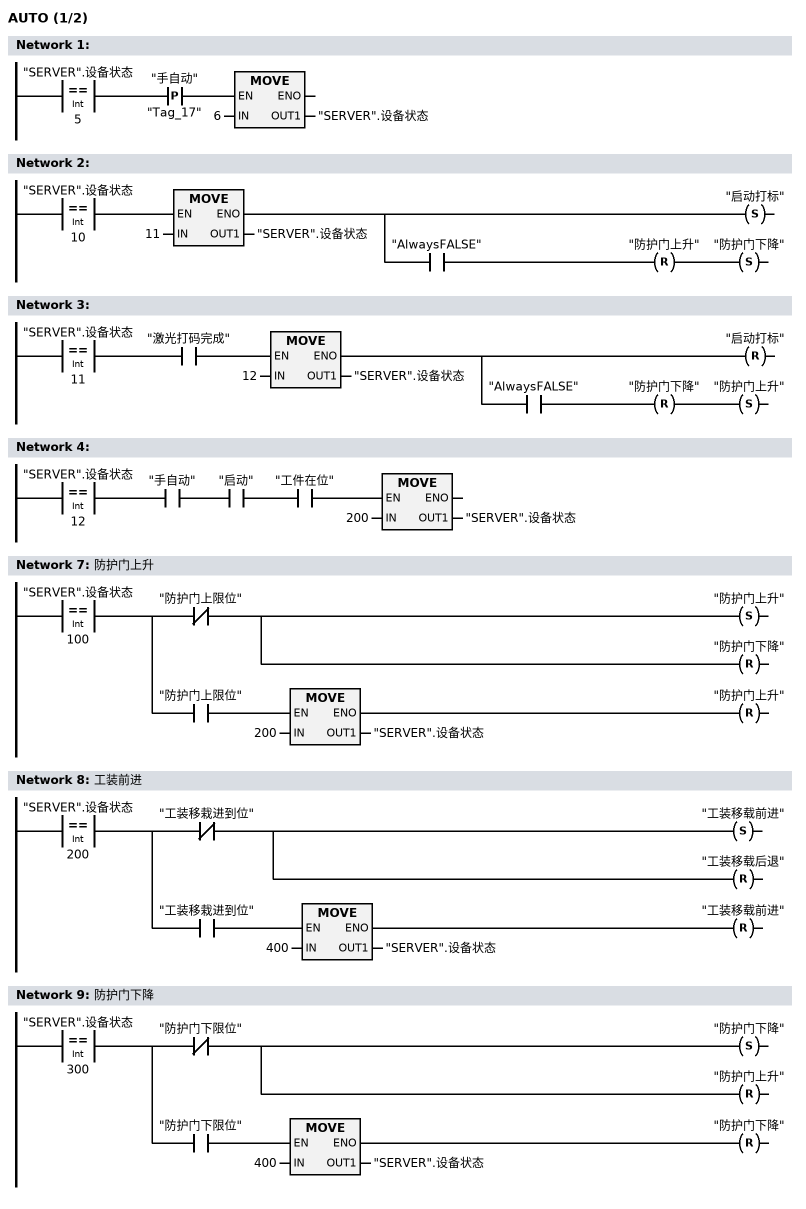
   RUNG wire#powerrail
      { S7_Templates := "SrcType := Int" } EQ_Contact(in1 := "SERVER".设备状态, in2 := 5)
      P_Contact(operand := "手自动", bit := "Tag_17")
      Move(in := 6, out1 => "SERVER".设备状态)
   END_RUNG
   // the same network as SCL:
   #_w1 := ("SERVER".设备状态 = 5) AND "手自动" AND NOT "Tag_17";   // rising edge of "手自动"
   "Tag_17" := "手自动";
   IF #_w1 THEN "SERVER".设备状态 := 6; END_IF;
END_REGION

REGION Network 2
   RUNG wire#powerrail
      { S7_Templates := "SrcType := Int" } EQ_Contact(in1 := "SERVER".设备状态, in2 := 10)
      Move(in := 11, out1 => "SERVER".设备状态)
      wire#w1
      S_Coil( "启动打标" )
   END_RUNG
   RUNG wire#w1
      Contact( "AlwaysFALSE" )
      R_Coil( "防护门上升" )
      S_Coil( "防护门下降" )
   END_RUNG
   // the same network as SCL:
   #_w1 := "SERVER".设备状态 = 10;
   IF #_w1 THEN
       "SERVER".设备状态 := 11;
       "启动打标" := TRUE;
   END_IF;
   IF #_w1 AND "AlwaysFALSE" THEN
       "防护门上升" := FALSE;
       "防护门下降" := TRUE;
   END_IF;
END_REGION

REGION Network 3
   RUNG wire#powerrail
      { S7_Templates := "SrcType := Int" } EQ_Contact(in1 := "SERVER".设备状态, in2 := 11)
      Contact( "激光打码完成" )
      Move(in := 12, out1 => "SERVER".设备状态)
      wire#w1
      R_Coil( "启动打标" )
   END_RUNG
   RUNG wire#w1
      Contact( "AlwaysFALSE" )
      R_Coil( "防护门下降" )
      S_Coil( "防护门上升" )
   END_RUNG
   // the same network as SCL:
   #_w1 := ("SERVER".设备状态 = 11) AND "激光打码完成";
   IF #_w1 THEN
       "SERVER".设备状态 := 12;
       "启动打标" := FALSE;
   END_IF;
   IF #_w1 AND "AlwaysFALSE" THEN
       "防护门下降" := FALSE;
       "防护门上升" := TRUE;
   END_IF;
END_REGION

REGION Network 4
   RUNG wire#powerrail
      { S7_Templates := "SrcType := Int" } EQ_Contact(in1 := "SERVER".设备状态, in2 := 12)
      Contact( "手自动" )
      Contact( "启动" )
      Contact( "工件在位" )
      Move(in := 200, out1 => "SERVER".设备状态)
   END_RUNG
   // the same network as SCL:
   IF ("SERVER".设备状态 = 12) AND "手自动" AND "启动" AND "工件在位" THEN "SERVER".设备状态 := 200; END_IF;
END_REGION

REGION Network 7: 防护门上升
   RUNG wire#powerrail
      { S7_Templates := "SrcType := Int" } EQ_Contact(in1 := "SERVER".设备状态, in2 := 100)
      wire#w1
      I_Contact( "防护门上限位" )
      wire#w2
      S_Coil( "防护门上升" )
   END_RUNG
   RUNG wire#w2
      R_Coil( "防护门下降" )
   END_RUNG
   RUNG wire#w1
      Contact( "防护门上限位" )
      Move(in := 200, out1 => "SERVER".设备状态)
      R_Coil( "防护门上升" )
   END_RUNG
   // the same network as SCL:
   #_w1 := "SERVER".设备状态 = 100;
   IF #_w1 AND NOT "防护门上限位" THEN
       "防护门上升" := TRUE;
       "防护门下降" := FALSE;
   END_IF;
   IF #_w1 AND "防护门上限位" THEN
       "SERVER".设备状态 := 200;
       "防护门上升" := FALSE;
   END_IF;
END_REGION

REGION Network 8: 工装前进
   RUNG wire#powerrail
      { S7_Templates := "SrcType := Int" } EQ_Contact(in1 := "SERVER".设备状态, in2 := 200)
      wire#w1
      I_Contact( "工装移栽进到位" )
      wire#w2
      S_Coil( "工装移载前进" )
   END_RUNG
   RUNG wire#w2
      R_Coil( "工装移载后退" )
   END_RUNG
   RUNG wire#w1
      Contact( "工装移栽进到位" )
      Move(in := 400, out1 => "SERVER".设备状态)
      R_Coil( "工装移载前进" )
   END_RUNG
   // the same network as SCL:
   #_w1 := "SERVER".设备状态 = 200;
   IF #_w1 AND NOT "工装移栽进到位" THEN
       "工装移载前进" := TRUE;
       "工装移载后退" := FALSE;
   END_IF;
   IF #_w1 AND "工装移栽进到位" THEN
       "SERVER".设备状态 := 400;
       "工装移载前进" := FALSE;
   END_IF;
END_REGION

REGION Network 9: 防护门下降
   RUNG wire#powerrail
      { S7_Templates := "SrcType := Int" } EQ_Contact(in1 := "SERVER".设备状态, in2 := 300)
      wire#w1
      I_Contact( "防护门下限位" )
      wire#w2
      S_Coil( "防护门下降" )
   END_RUNG
   RUNG wire#w2
      R_Coil( "防护门上升" )
   END_RUNG
   RUNG wire#w1
      Contact( "防护门下限位" )
      Move(in := 400, out1 => "SERVER".设备状态)
      R_Coil( "防护门下降" )
   END_RUNG
   // the same network as SCL:
   #_w1 := "SERVER".设备状态 = 300;
   IF #_w1 AND NOT "防护门下限位" THEN
       "防护门下降" := TRUE;
       "防护门上升" := FALSE;
   END_IF;
   IF #_w1 AND "防护门下限位" THEN
       "SERVER".设备状态 := 400;
       "防护门下降" := FALSE;
   END_IF;
END_REGION

REGION Network 10: 激光打标
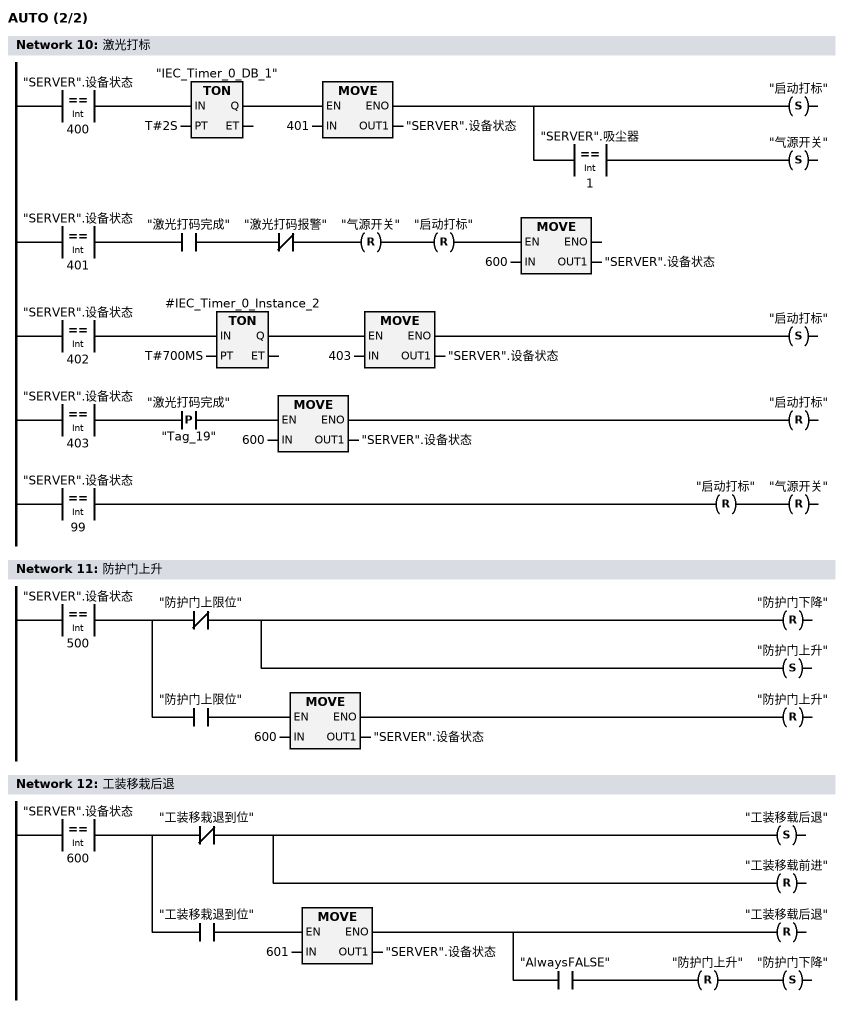
   "IEC_Timer_0_DB_1".TON(IN := "SERVER".设备状态 = 400, PT := T#2S);
   IF "IEC_Timer_0_DB_1".Q THEN
       "SERVER".设备状态 := 401;
       "启动打标" := TRUE;
   END_IF;
   IF "IEC_Timer_0_DB_1".Q AND ("SERVER".吸尘器 = 1) THEN "气源开关" := TRUE; END_IF;
   IF ("SERVER".设备状态 = 401) AND "激光打码完成" AND NOT "激光打码报警" THEN
       "气源开关" := FALSE;
       "启动打标" := FALSE;
       "SERVER".设备状态 := 600;
   END_IF;
   #IEC_Timer_0_Instance_2(IN := "SERVER".设备状态 = 402, PT := T#700MS);   // TON
   IF #IEC_Timer_0_Instance_2.Q THEN
       "SERVER".设备状态 := 403;
       "启动打标" := TRUE;
   END_IF;
   #_w1 := ("SERVER".设备状态 = 403) AND "激光打码完成" AND NOT "Tag_19";   // rising edge of "激光打码完成"
   "Tag_19" := "激光打码完成";
   IF #_w1 THEN
       "SERVER".设备状态 := 600;
       "启动打标" := FALSE;
   END_IF;
   IF "SERVER".设备状态 = 99 THEN
       "启动打标" := FALSE;
       "气源开关" := FALSE;
   END_IF;
END_REGION

REGION Network 11: 防护门上升
   RUNG wire#powerrail
      { S7_Templates := "SrcType := Int" } EQ_Contact(in1 := "SERVER".设备状态, in2 := 500)
      wire#w1
      I_Contact( "防护门上限位" )
      wire#w2
      R_Coil( "防护门下降" )
   END_RUNG
   RUNG wire#w2
      S_Coil( "防护门上升" )
   END_RUNG
   RUNG wire#w1
      Contact( "防护门上限位" )
      Move(in := 600, out1 => "SERVER".设备状态)
      R_Coil( "防护门上升" )
   END_RUNG
   // the same network as SCL:
   #_w1 := "SERVER".设备状态 = 500;
   IF #_w1 AND NOT "防护门上限位" THEN
       "防护门下降" := FALSE;
       "防护门上升" := TRUE;
   END_IF;
   IF #_w1 AND "防护门上限位" THEN
       "SERVER".设备状态 := 600;
       "防护门上升" := FALSE;
   END_IF;
END_REGION

REGION Network 12: 工装移栽后退
   RUNG wire#powerrail
      { S7_Templates := "SrcType := Int" } EQ_Contact(in1 := "SERVER".设备状态, in2 := 600)
      wire#w1
      I_Contact( "工装移栽退到位" )
      wire#w2
      S_Coil( "工装移载后退" )
   END_RUNG
   RUNG wire#w2
      R_Coil( "工装移载前进" )
   END_RUNG
   RUNG wire#w1
      Contact( "工装移栽退到位" )
      Move(in := 601, out1 => "SERVER".设备状态)
      wire#w3
      R_Coil( "工装移载后退" )
   END_RUNG
   RUNG wire#w3
      Contact( "AlwaysFALSE" )
      R_Coil( "防护门上升" )
      S_Coil( "防护门下降" )
   END_RUNG
   // the same network as SCL:
   #_w1 := "SERVER".设备状态 = 600;
   IF #_w1 AND NOT "工装移栽退到位" THEN
       "工装移载后退" := TRUE;
       "工装移载前进" := FALSE;
   END_IF;
   #_w2 := #_w1 AND "工装移栽退到位";
   IF #_w2 THEN
       "SERVER".设备状态 := 601;
       "工装移载后退" := FALSE;
   END_IF;
   IF #_w2 AND "AlwaysFALSE" THEN
       "防护门上升" := FALSE;
       "防护门下降" := TRUE;
   END_IF;
END_REGION
END_FUNCTION_BLOCK

FUNCTION_BLOCK "1# jixieshou"   // FB4, LAD
{ S7_Optimized_Access := 'TRUE' }
VERSION : 0.1
   VAR
      temp_1 : Bool;
      temp_2 : Bool;
      "Step-1" : Int;
      IEC_Timer_0_Instance : TON_TIME;
      IEC_Timer_0_Instance_1 : TON_TIME;
      IEC_Timer_0_Instance_2 : TON_TIME;
      IEC_Timer_0_Instance_3 : TON_TIME;
      IEC_Timer_0_Instance_4 : TON_TIME;
      IEC_Timer_0_Instance_5 : TON_TIME;
      IEC_Timer_0_Instance_6 : TON_TIME;
   END_VAR
   VAR_TEMP   // added for the SCL form of the ladder/FBD networks
      _w1 : Bool;
      _w2 : Bool;
   END_VAR
BEGIN

REGION Network 1
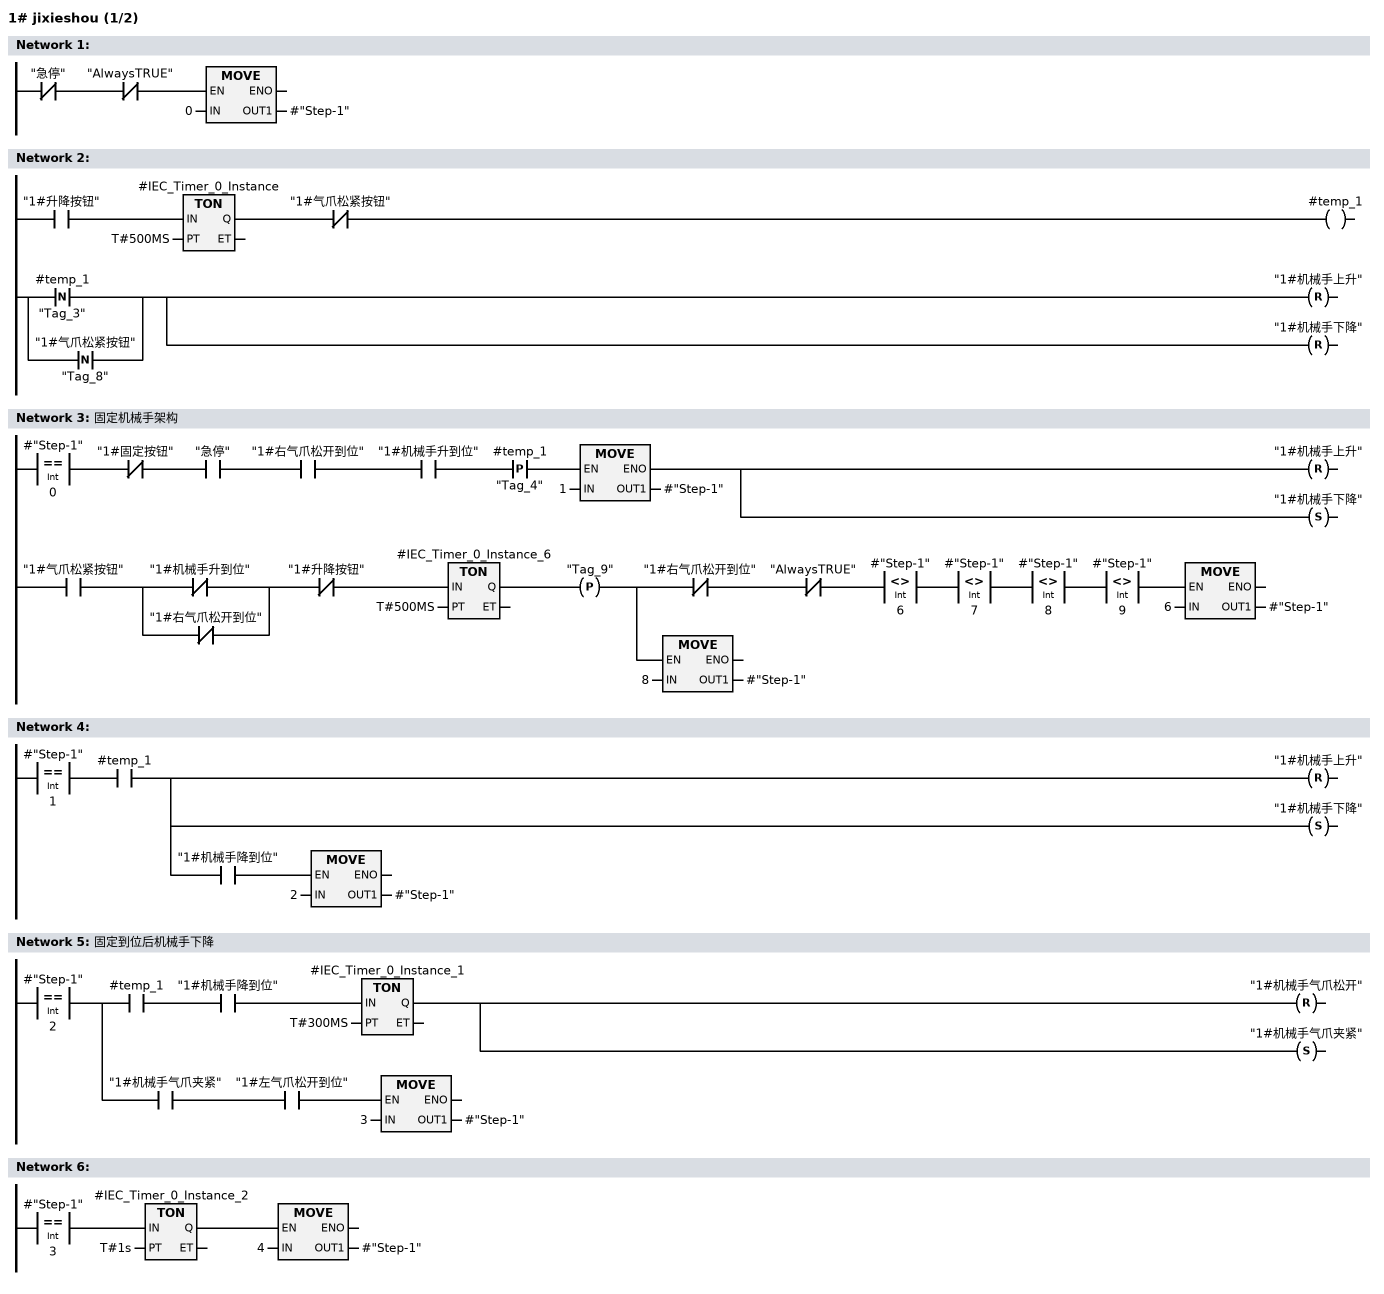
   RUNG wire#powerrail
      I_Contact( "急停" )
      I_Contact( "AlwaysTRUE" )
      Move(in := 0, out1 => #"Step-1")
   END_RUNG
   // the same network as SCL:
   IF NOT "急停" AND NOT "AlwaysTRUE" THEN #"Step-1" := 0; END_IF;
END_REGION

REGION Network 2
   #IEC_Timer_0_Instance(IN := "1#升降按钮", PT := T#500MS);   // TON
   #temp_1 := #IEC_Timer_0_Instance.Q AND NOT "1#气爪松紧按钮";
   #_w1 := NOT #temp_1 AND "Tag_3";   // falling edge of #temp_1
   "Tag_3" := #temp_1;
   #_w2 := NOT "1#气爪松紧按钮" AND "Tag_8";   // falling edge of "1#气爪松紧按钮"
   "Tag_8" := "1#气爪松紧按钮";
   IF #_w1 OR #_w2 THEN
       "1#机械手上升" := FALSE;
       "1#机械手下降" := FALSE;
   END_IF;
END_REGION

REGION Network 3: 固定机械手架构
   #_w1 := (#"Step-1" = 0) AND NOT "1#固定按钮" AND "急停" AND "1#右气爪松开到位" AND "1#机械手升到位" AND #temp_1 AND NOT "Tag_4";   // rising edge of #temp_1
   "Tag_4" := #temp_1;
   IF #_w1 THEN
       #"Step-1" := 1;
       "1#机械手上升" := FALSE;
       "1#机械手下降" := TRUE;
   END_IF;
   #IEC_Timer_0_Instance_6(IN := "1#气爪松紧按钮" AND (NOT "1#机械手升到位" OR NOT "1#右气爪松开到位") AND NOT "1#升降按钮",   // TON
                           PT := T#500MS);
   #_w2 := #IEC_Timer_0_Instance_6.Q AND NOT "Tag_9";   // rising edge
   "Tag_9" := #IEC_Timer_0_Instance_6.Q;
   IF #_w2 AND NOT "1#右气爪松开到位" AND NOT "AlwaysTRUE" AND (#"Step-1" <> 6) AND (#"Step-1" <> 7) AND (#"Step-1" <> 8) AND (#"Step-1" <> 9) THEN
       #"Step-1" := 6;
   END_IF;
   IF #_w2 THEN #"Step-1" := 8; END_IF;
END_REGION

REGION Network 4
   RUNG wire#powerrail
      { S7_Templates := "SrcType := Int" } EQ_Contact(in1 := #"Step-1", in2 := 1)
      Contact( #temp_1 )
      wire#w1
      R_Coil( "1#机械手上升" )
   END_RUNG
   RUNG wire#w1
      S_Coil( "1#机械手下降" )
   END_RUNG
   RUNG wire#w1
      Contact( "1#机械手降到位" )
      Move(in := 2, out1 => #"Step-1")
   END_RUNG
   // the same network as SCL:
   #_w1 := (#"Step-1" = 1) AND #temp_1;
   IF #_w1 THEN
       "1#机械手上升" := FALSE;
       "1#机械手下降" := TRUE;
   END_IF;
   IF #_w1 AND "1#机械手降到位" THEN #"Step-1" := 2; END_IF;
END_REGION

REGION Network 5: 固定到位后机械手下降
   #_w1 := #"Step-1" = 2;
   #IEC_Timer_0_Instance_1(IN := #_w1 AND #temp_1 AND "1#机械手降到位", PT := T#300MS);   // TON
   IF #IEC_Timer_0_Instance_1.Q THEN
       "1#机械手气爪松开" := FALSE;
       "1#机械手气爪夹紧" := TRUE;
   END_IF;
   IF #_w1 AND "1#机械手气爪夹紧" AND "1#左气爪松开到位" THEN #"Step-1" := 3; END_IF;
END_REGION

REGION Network 6
   #IEC_Timer_0_Instance_2(IN := #"Step-1" = 3, PT := T#1s);   // TON
   IF #IEC_Timer_0_Instance_2.Q THEN #"Step-1" := 4; END_IF;
END_REGION

REGION Network 7: 下降到位后气爪夹紧
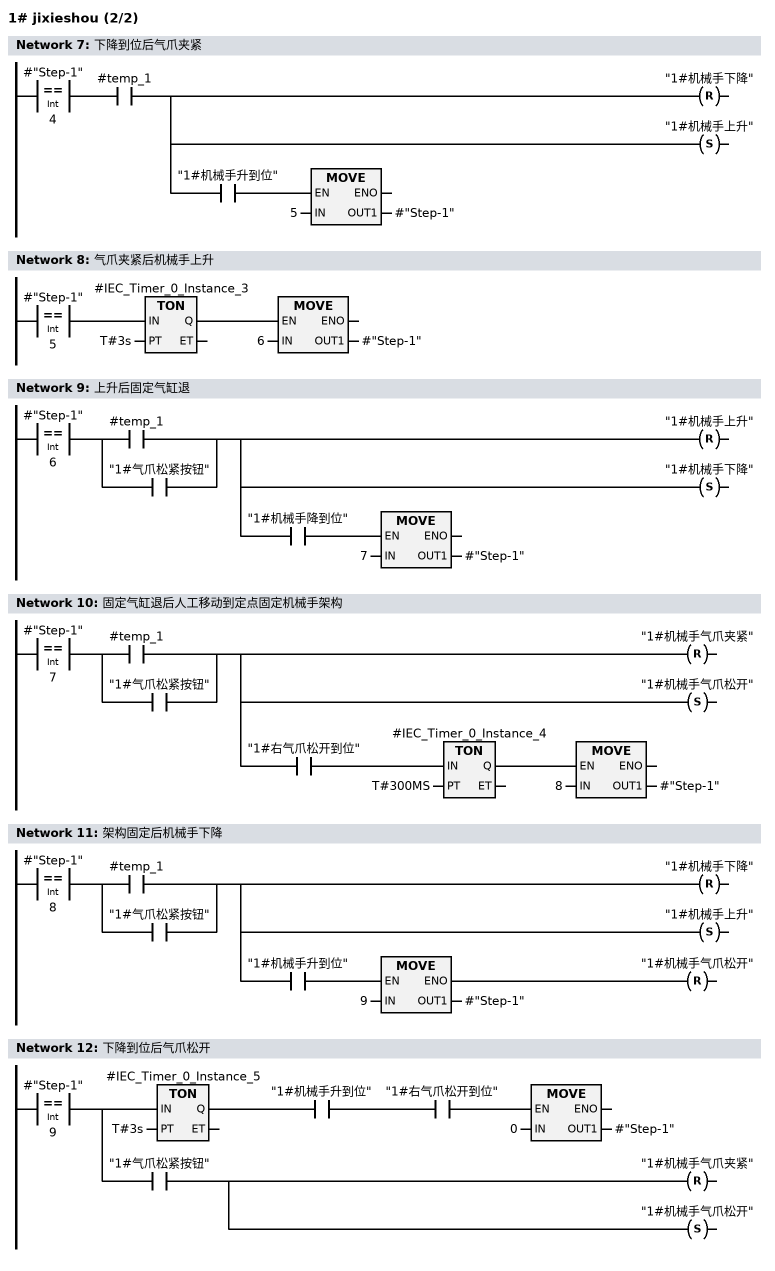
   RUNG wire#powerrail
      { S7_Templates := "SrcType := Int" } EQ_Contact(in1 := #"Step-1", in2 := 4)
      Contact( #temp_1 )
      wire#w1
      R_Coil( "1#机械手下降" )
   END_RUNG
   RUNG wire#w1
      S_Coil( "1#机械手上升" )
   END_RUNG
   RUNG wire#w1
      Contact( "1#机械手升到位" )
      Move(in := 5, out1 => #"Step-1")
   END_RUNG
   // the same network as SCL:
   #_w1 := (#"Step-1" = 4) AND #temp_1;
   IF #_w1 THEN
       "1#机械手下降" := FALSE;
       "1#机械手上升" := TRUE;
   END_IF;
   IF #_w1 AND "1#机械手升到位" THEN #"Step-1" := 5; END_IF;
END_REGION

REGION Network 8: 气爪夹紧后机械手上升
   #IEC_Timer_0_Instance_3(IN := #"Step-1" = 5, PT := T#3s);   // TON
   IF #IEC_Timer_0_Instance_3.Q THEN #"Step-1" := 6; END_IF;
END_REGION

REGION Network 9: 上升后固定气缸退
   RUNG wire#powerrail
      { S7_Templates := "SrcType := Int" } EQ_Contact(in1 := #"Step-1", in2 := 6)
      wire#w1
      Contact( #temp_1 )
      wire#w2
      R_Coil( "1#机械手上升" )
   END_RUNG
   RUNG wire#w1
      Contact( "1#气爪松紧按钮" )
   END_RUNG wire#w2
   RUNG wire#w2
      S_Coil( "1#机械手下降" )
   END_RUNG
   RUNG wire#w2
      Contact( "1#机械手降到位" )
      Move(in := 7, out1 => #"Step-1")
   END_RUNG
   // the same network as SCL:
   #_w1 := (#"Step-1" = 6) AND (#temp_1 OR "1#气爪松紧按钮");
   IF #_w1 THEN
       "1#机械手上升" := FALSE;
       "1#机械手下降" := TRUE;
   END_IF;
   IF #_w1 AND "1#机械手降到位" THEN #"Step-1" := 7; END_IF;
END_REGION

REGION Network 10: 固定气缸退后人工移动到定点固定机械手架构
   #_w1 := (#"Step-1" = 7) AND (#temp_1 OR "1#气爪松紧按钮");
   IF #_w1 THEN
       "1#机械手气爪夹紧" := FALSE;
       "1#机械手气爪松开" := TRUE;
   END_IF;
   #IEC_Timer_0_Instance_4(IN := #_w1 AND "1#右气爪松开到位", PT := T#300MS);   // TON
   IF #IEC_Timer_0_Instance_4.Q THEN #"Step-1" := 8; END_IF;
END_REGION

REGION Network 11: 架构固定后机械手下降
   RUNG wire#powerrail
      { S7_Templates := "SrcType := Int" } EQ_Contact(in1 := #"Step-1", in2 := 8)
      wire#w1
      Contact( #temp_1 )
      wire#w2
      R_Coil( "1#机械手下降" )
   END_RUNG
   RUNG wire#w1
      Contact( "1#气爪松紧按钮" )
   END_RUNG wire#w2
   RUNG wire#w2
      S_Coil( "1#机械手上升" )
   END_RUNG
   RUNG wire#w2
      Contact( "1#机械手升到位" )
      Move(in := 9, out1 => #"Step-1")
      R_Coil( "1#机械手气爪松开" )
   END_RUNG
   // the same network as SCL:
   #_w1 := (#"Step-1" = 8) AND (#temp_1 OR "1#气爪松紧按钮");
   IF #_w1 THEN
       "1#机械手下降" := FALSE;
       "1#机械手上升" := TRUE;
   END_IF;
   IF #_w1 AND "1#机械手升到位" THEN
       #"Step-1" := 9;
       "1#机械手气爪松开" := FALSE;
   END_IF;
END_REGION

REGION Network 12: 下降到位后气爪松开
   #_w1 := #"Step-1" = 9;
   #IEC_Timer_0_Instance_5(IN := #_w1, PT := T#3s);   // TON
   IF #IEC_Timer_0_Instance_5.Q AND "1#机械手升到位" AND "1#右气爪松开到位" THEN #"Step-1" := 0; END_IF;
   IF #_w1 AND "1#气爪松紧按钮" THEN
       "1#机械手气爪夹紧" := FALSE;
       "1#机械手气爪松开" := TRUE;
   END_IF;
END_REGION
END_FUNCTION_BLOCK

FUNCTION_BLOCK "2#jixieshou"   // FB5, LAD
{ S7_Optimized_Access := 'TRUE' }
VERSION : 0.1
   VAR
      temp_1 : Bool;
      "Step-2" : Int;
      IEC_Timer_0_Instance : TON_TIME;
      IEC_Timer_0_Instance_1 : TON_TIME;
      IEC_Timer_0_Instance_2 : TON_TIME;
      IEC_Timer_0_Instance_3 : TON_TIME;
      IEC_Timer_0_Instance_4 : TON_TIME;
      IEC_Timer_0_Instance_5 : TON_TIME;
      IEC_Timer_0_Instance_6 : TON_TIME;
   END_VAR
   VAR_TEMP   // added for the SCL form of the ladder/FBD networks
      _w1 : Bool;
      _w2 : Bool;
   END_VAR
BEGIN

REGION Network 1
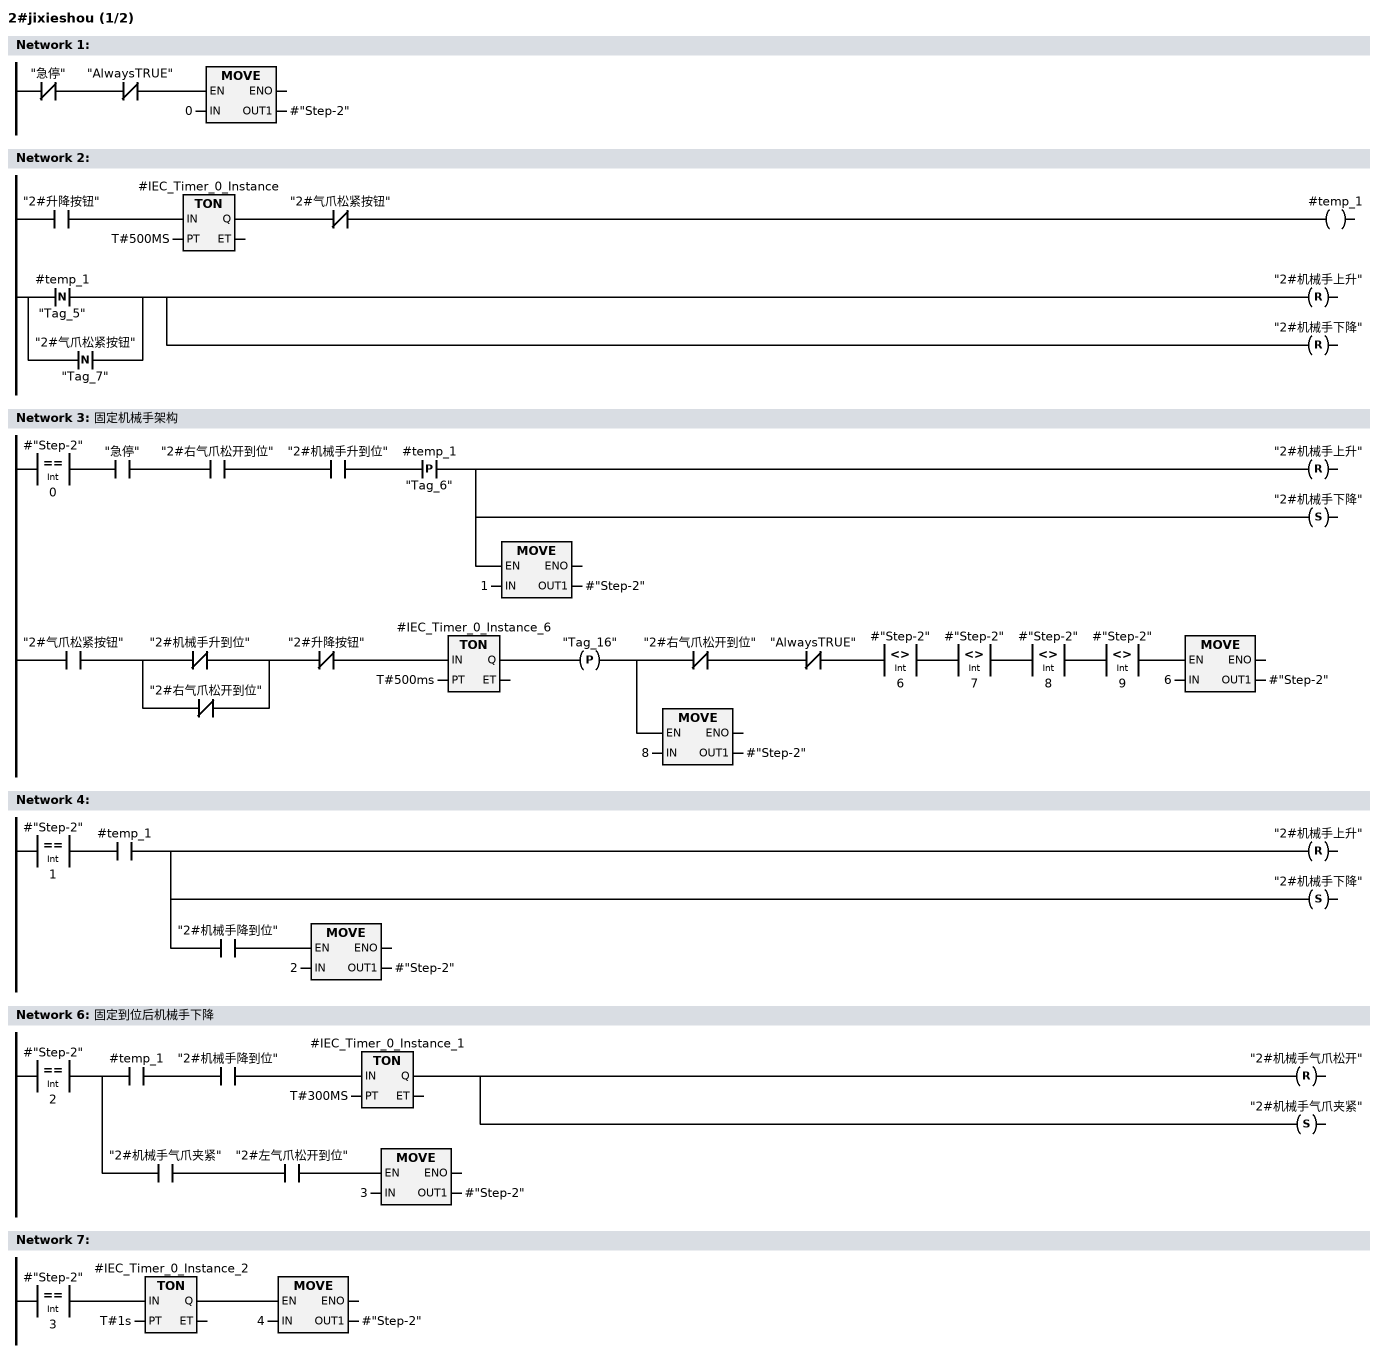
   RUNG wire#powerrail
      I_Contact( "急停" )
      I_Contact( "AlwaysTRUE" )
      Move(in := 0, out1 => #"Step-2")
   END_RUNG
   // the same network as SCL:
   IF NOT "急停" AND NOT "AlwaysTRUE" THEN #"Step-2" := 0; END_IF;
END_REGION

REGION Network 2
   #IEC_Timer_0_Instance(IN := "2#升降按钮", PT := T#500MS);   // TON
   #temp_1 := #IEC_Timer_0_Instance.Q AND NOT "2#气爪松紧按钮";
   #_w1 := NOT #temp_1 AND "Tag_5";   // falling edge of #temp_1
   "Tag_5" := #temp_1;
   #_w2 := NOT "2#气爪松紧按钮" AND "Tag_7";   // falling edge of "2#气爪松紧按钮"
   "Tag_7" := "2#气爪松紧按钮";
   IF #_w1 OR #_w2 THEN
       "2#机械手上升" := FALSE;
       "2#机械手下降" := FALSE;
   END_IF;
END_REGION

REGION Network 3: 固定机械手架构
   #_w1 := (#"Step-2" = 0) AND "急停" AND "2#右气爪松开到位" AND "2#机械手升到位" AND #temp_1 AND NOT "Tag_6";   // rising edge of #temp_1
   "Tag_6" := #temp_1;
   IF #_w1 THEN
       "2#机械手上升" := FALSE;
       "2#机械手下降" := TRUE;
       #"Step-2" := 1;
   END_IF;
   #IEC_Timer_0_Instance_6(IN := "2#气爪松紧按钮" AND (NOT "2#机械手升到位" OR NOT "2#右气爪松开到位") AND NOT "2#升降按钮",   // TON
                           PT := T#500ms);
   #_w2 := #IEC_Timer_0_Instance_6.Q AND NOT "Tag_16";   // rising edge
   "Tag_16" := #IEC_Timer_0_Instance_6.Q;
   IF #_w2 AND NOT "2#右气爪松开到位" AND NOT "AlwaysTRUE" AND (#"Step-2" <> 6) AND (#"Step-2" <> 7) AND (#"Step-2" <> 8) AND (#"Step-2" <> 9) THEN
       #"Step-2" := 6;
   END_IF;
   IF #_w2 THEN #"Step-2" := 8; END_IF;
END_REGION

REGION Network 4
   RUNG wire#powerrail
      { S7_Templates := "SrcType := Int" } EQ_Contact(in1 := #"Step-2", in2 := 1)
      Contact( #temp_1 )
      wire#w1
      R_Coil( "2#机械手上升" )
   END_RUNG
   RUNG wire#w1
      S_Coil( "2#机械手下降" )
   END_RUNG
   RUNG wire#w1
      Contact( "2#机械手降到位" )
      Move(in := 2, out1 => #"Step-2")
   END_RUNG
   // the same network as SCL:
   #_w1 := (#"Step-2" = 1) AND #temp_1;
   IF #_w1 THEN
       "2#机械手上升" := FALSE;
       "2#机械手下降" := TRUE;
   END_IF;
   IF #_w1 AND "2#机械手降到位" THEN #"Step-2" := 2; END_IF;
END_REGION

REGION Network 6: 固定到位后机械手下降
   #_w1 := #"Step-2" = 2;
   #IEC_Timer_0_Instance_1(IN := #_w1 AND #temp_1 AND "2#机械手降到位", PT := T#300MS);   // TON
   IF #IEC_Timer_0_Instance_1.Q THEN
       "2#机械手气爪松开" := FALSE;
       "2#机械手气爪夹紧" := TRUE;
   END_IF;
   IF #_w1 AND "2#机械手气爪夹紧" AND "2#左气爪松开到位" THEN #"Step-2" := 3; END_IF;
END_REGION

REGION Network 7
   #IEC_Timer_0_Instance_2(IN := #"Step-2" = 3, PT := T#1s);   // TON
   IF #IEC_Timer_0_Instance_2.Q THEN #"Step-2" := 4; END_IF;
END_REGION

REGION Network 8: 下降到位后气爪夹紧
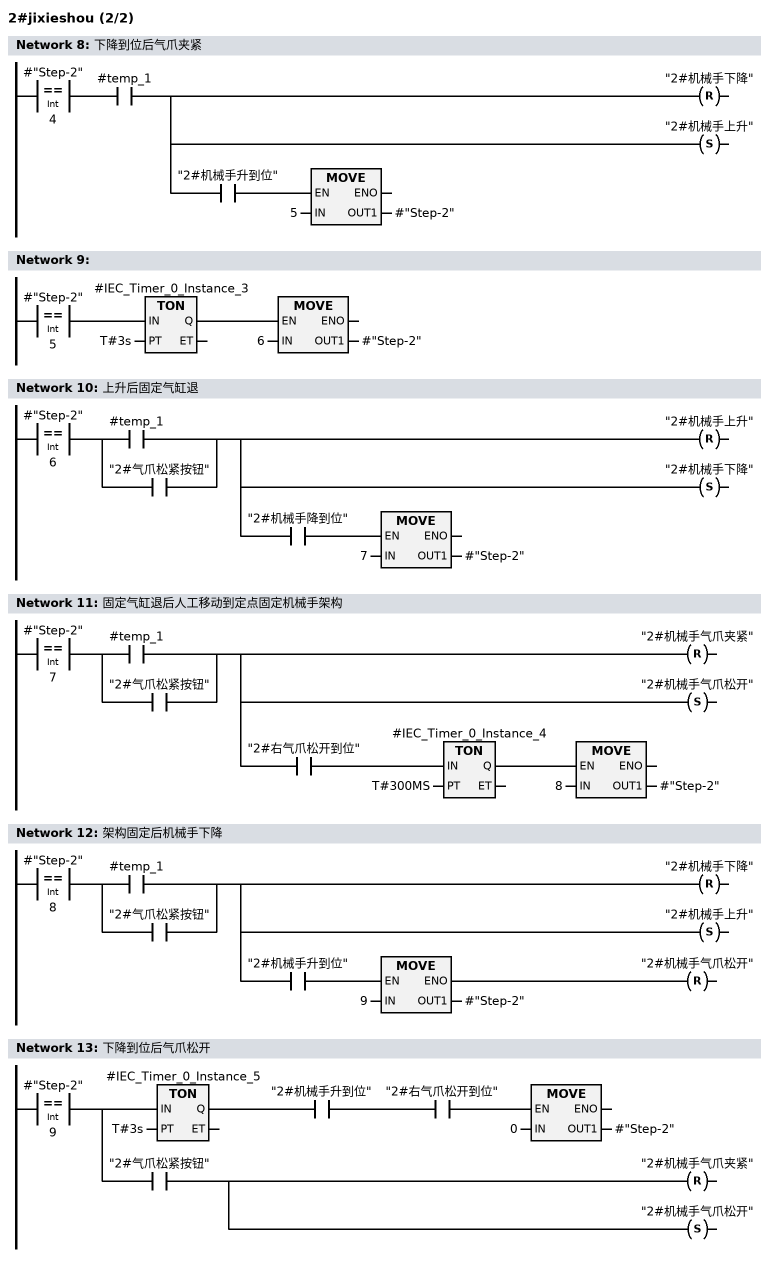
   RUNG wire#powerrail
      { S7_Templates := "SrcType := Int" } EQ_Contact(in1 := #"Step-2", in2 := 4)
      Contact( #temp_1 )
      wire#w1
      R_Coil( "2#机械手下降" )
   END_RUNG
   RUNG wire#w1
      S_Coil( "2#机械手上升" )
   END_RUNG
   RUNG wire#w1
      Contact( "2#机械手升到位" )
      Move(in := 5, out1 => #"Step-2")
   END_RUNG
   // the same network as SCL:
   #_w1 := (#"Step-2" = 4) AND #temp_1;
   IF #_w1 THEN
       "2#机械手下降" := FALSE;
       "2#机械手上升" := TRUE;
   END_IF;
   IF #_w1 AND "2#机械手升到位" THEN #"Step-2" := 5; END_IF;
END_REGION

REGION Network 9
   #IEC_Timer_0_Instance_3(IN := #"Step-2" = 5, PT := T#3s);   // TON
   IF #IEC_Timer_0_Instance_3.Q THEN #"Step-2" := 6; END_IF;
END_REGION

REGION Network 10: 上升后固定气缸退
   RUNG wire#powerrail
      { S7_Templates := "SrcType := Int" } EQ_Contact(in1 := #"Step-2", in2 := 6)
      wire#w1
      Contact( #temp_1 )
      wire#w2
      R_Coil( "2#机械手上升" )
   END_RUNG
   RUNG wire#w1
      Contact( "2#气爪松紧按钮" )
   END_RUNG wire#w2
   RUNG wire#w2
      S_Coil( "2#机械手下降" )
   END_RUNG
   RUNG wire#w2
      Contact( "2#机械手降到位" )
      Move(in := 7, out1 => #"Step-2")
   END_RUNG
   // the same network as SCL:
   #_w1 := (#"Step-2" = 6) AND (#temp_1 OR "2#气爪松紧按钮");
   IF #_w1 THEN
       "2#机械手上升" := FALSE;
       "2#机械手下降" := TRUE;
   END_IF;
   IF #_w1 AND "2#机械手降到位" THEN #"Step-2" := 7; END_IF;
END_REGION

REGION Network 11: 固定气缸退后人工移动到定点固定机械手架构
   #_w1 := (#"Step-2" = 7) AND (#temp_1 OR "2#气爪松紧按钮");
   IF #_w1 THEN
       "2#机械手气爪夹紧" := FALSE;
       "2#机械手气爪松开" := TRUE;
   END_IF;
   #IEC_Timer_0_Instance_4(IN := #_w1 AND "2#右气爪松开到位", PT := T#300MS);   // TON
   IF #IEC_Timer_0_Instance_4.Q THEN #"Step-2" := 8; END_IF;
END_REGION

REGION Network 12: 架构固定后机械手下降
   RUNG wire#powerrail
      { S7_Templates := "SrcType := Int" } EQ_Contact(in1 := #"Step-2", in2 := 8)
      wire#w1
      Contact( #temp_1 )
      wire#w2
      R_Coil( "2#机械手下降" )
   END_RUNG
   RUNG wire#w1
      Contact( "2#气爪松紧按钮" )
   END_RUNG wire#w2
   RUNG wire#w2
      S_Coil( "2#机械手上升" )
   END_RUNG
   RUNG wire#w2
      Contact( "2#机械手升到位" )
      Move(in := 9, out1 => #"Step-2")
      R_Coil( "2#机械手气爪松开" )
   END_RUNG
   // the same network as SCL:
   #_w1 := (#"Step-2" = 8) AND (#temp_1 OR "2#气爪松紧按钮");
   IF #_w1 THEN
       "2#机械手下降" := FALSE;
       "2#机械手上升" := TRUE;
   END_IF;
   IF #_w1 AND "2#机械手升到位" THEN
       #"Step-2" := 9;
       "2#机械手气爪松开" := FALSE;
   END_IF;
END_REGION

REGION Network 13: 下降到位后气爪松开
   #_w1 := #"Step-2" = 9;
   #IEC_Timer_0_Instance_5(IN := #_w1, PT := T#3s);   // TON
   IF #IEC_Timer_0_Instance_5.Q AND "2#机械手升到位" AND "2#右气爪松开到位" THEN #"Step-2" := 0; END_IF;
   IF #_w1 AND "2#气爪松紧按钮" THEN
       "2#机械手气爪夹紧" := FALSE;
       "2#机械手气爪松开" := TRUE;
   END_IF;
END_REGION
END_FUNCTION_BLOCK

ORGANIZATION_BLOCK "Main"   // OB1, LAD, ProgramCycle
TITLE = "Main Program Sweep (Cycle)"
{ S7_Optimized_Access := 'TRUE' }
VERSION : 0.1
   VAR_INPUT
      Initial_Call : Bool;   // Initial call of this OB
      Remanence : Bool;   // =True, if remanent data are available
   END_VAR
   VAR_TEMP   // added for the SCL form of the ladder/FBD networks
      _w1 : Bool;
   END_VAR
BEGIN

REGION Network 1
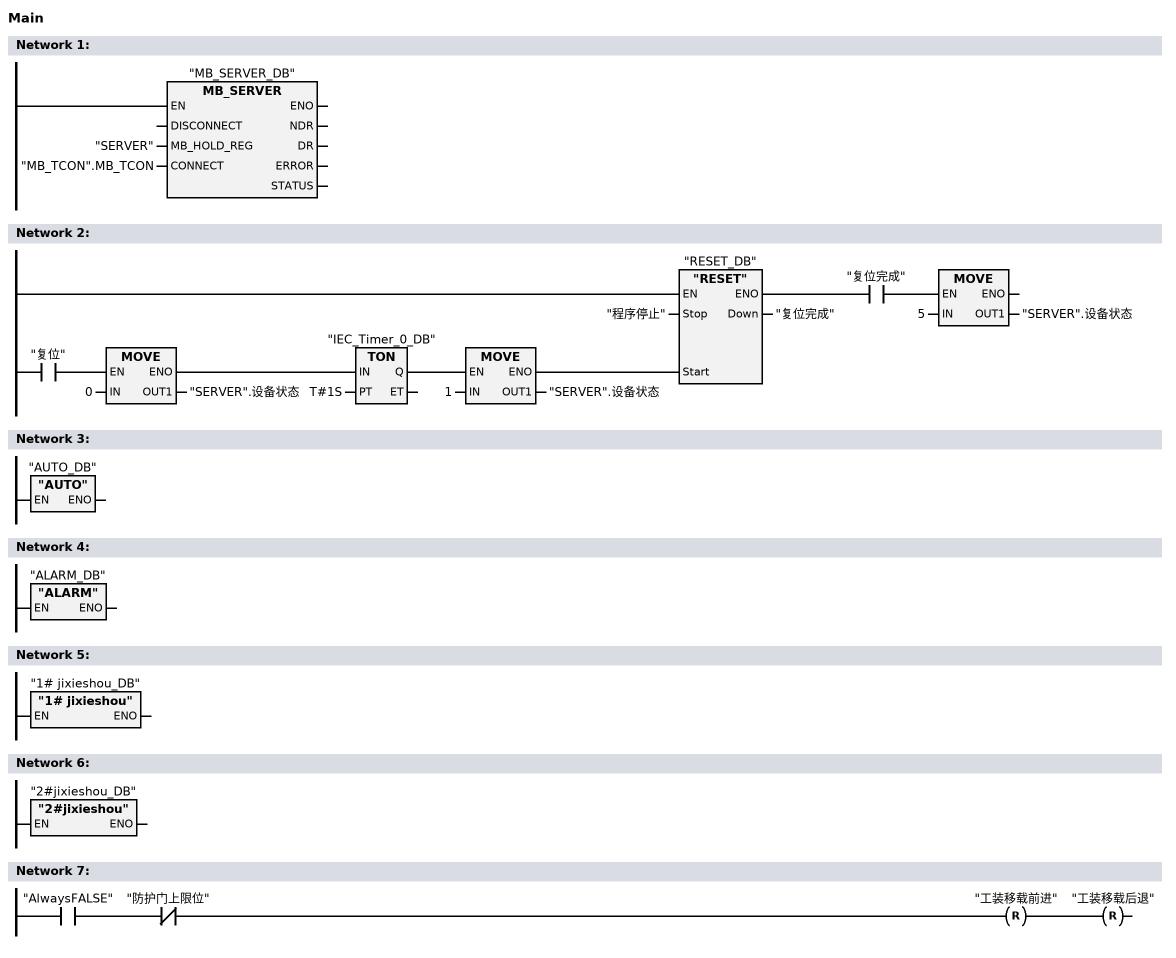
   "MB_SERVER_DB"(MB_HOLD_REG := "SERVER", CONNECT := "MB_TCON".MB_TCON);   // MB_SERVER
END_REGION

REGION Network 2
   IF "复位" THEN "SERVER".设备状态 := 0; END_IF;
   "IEC_Timer_0_DB".TON(IN := "复位", PT := T#1S);
   IF "IEC_Timer_0_DB".Q THEN "SERVER".设备状态 := 1; END_IF;
   "RESET_DB"(Stop := "程序停止", Start := "IEC_Timer_0_DB".Q, Down => "复位完成", ENO => #_w1);   // "RESET"
   IF #_w1 AND "复位完成" THEN "SERVER".设备状态 := 5; END_IF;
END_REGION

REGION Network 3
   RUNG wire#powerrail
      "AUTO_DB"()
   END_RUNG
   // the same network as SCL:
   "AUTO_DB"();   // "AUTO"
END_REGION

REGION Network 4
   RUNG wire#powerrail
      "ALARM_DB"()
   END_RUNG
   // the same network as SCL:
   "ALARM_DB"();   // "ALARM"
END_REGION

REGION Network 5
   RUNG wire#powerrail
      "1# jixieshou_DB"()
   END_RUNG
   // the same network as SCL:
   "1# jixieshou_DB"();   // "1# jixieshou"
END_REGION

REGION Network 6
   RUNG wire#powerrail
      "2#jixieshou_DB"()
   END_RUNG
   // the same network as SCL:
   "2#jixieshou_DB"();   // "2#jixieshou"
END_REGION

REGION Network 7
   RUNG wire#powerrail
      Contact( "AlwaysFALSE" )
      I_Contact( "防护门上限位" )
      R_Coil( "工装移载前进" )
      R_Coil( "工装移载后退" )
   END_RUNG
   // the same network as SCL:
   IF "AlwaysFALSE" AND NOT "防护门上限位" THEN
       "工装移载前进" := FALSE;
       "工装移载后退" := FALSE;
   END_IF;
END_REGION
END_ORGANIZATION_BLOCK